PROGRAM Emergency_Stop
VAR
END_VAR

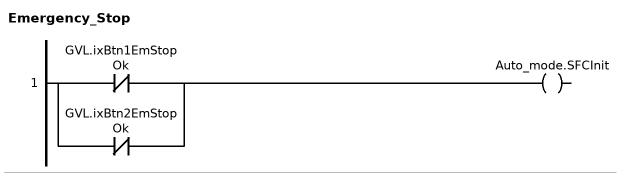
// NETWORK 1
Auto_mode.SFCInit := NOT GVL.ixBtn1EmStopOk OR NOT GVL.ixBtn2EmStopOk;

END_PROGRAM

(* stored: Version 1.1.0.1, ProductVersion 3.1.4024.12
   POU Emergency_Stop: Id {7083b58f-9232-4e0f-9c63-d6b78bc35624}, SpecialFunc None *)
